// SIMATIC S7-200 SMART project (STEP 7-Micro/WIN SMART), CPU SR40

SYMBOL_TABLE 系统符号
Always_On        SM0.0    // 始终接通
First_Scan_On    SM0.1    // 仅在第一个扫描周期时接通
HSC0_Ctrl        SMB37    // 组态和控制 HSC0
HSC0_CV          SMD38    // HSC0 新当前值
HSC0_PV          SMD42    // HSC0 新预设值
END_SYMBOL_TABLE

ORGANIZATION_BLOCK MAIN:OB1
TITLE=程序注释
BEGIN
Network 1
// 程序段注释
LD     First_Scan_On:SM0.1
CALL   HSC0_INIT:SBR1
Network 2
LD     Always_On:SM0.0
=      L60.0
LD     I0.1
=      L63.7
LD     L60.0
CALL   PWM0_RUN:SBR2, L63.7, 1000, 500, VB10
END_ORGANIZATION_BLOCK

SUBROUTINE_BLOCK HSC0_INIT:SBR1
TITLE=
BEGIN
Network 1
// 要在程序内启用该组态，请使用 SM0.1 或沿触发指令从 MAIN 程序块将该子程序调用一次。  
// 针对模式 0 组态 HC0； CV = 0； PV = 4000； 加计数； 
// 将中断 COUNT_EQ0 附加到事件 12 (HC0 的 CV = PV)。
// 启用中断并启动计数器。
// 
LD     Always_On:SM0.0
MOVB   16#F8, HSC0_Ctrl:SMB37 //置位控制位： 加计数； 已启用； 
MOVD   +0, HSC0_CV:SMD38     //装载 CV
MOVD   +4000, HSC0_PV:SMD42  //装载 PV
HDEF   0, 0
ATCH   COUNT_EQ0:INT1, 12    //中断 COUNT_EQ0：HC0 的 CV = PV
ENI
HSC    0
SI     Q0.1, 1
RI     Q0.2, 1
END_SUBROUTINE_BLOCK

// SBR2: protected block, not included

INTERRUPT_BLOCK COUNT_EQ0:INT1
TITLE=
BEGIN
Network 1
// (CV = PV) 步 1，3，HC0
// 编译 HC0 的动态参数； PV = 7000； 
// 将中断 HSC0_STEP1 附加到事件 12 (HC0 的 CV = PV)。
// 启动计数器。
// 
LD     Always_On:SM0.0
MOVB   16#A0, HSC0_Ctrl:SMB37 //置位控制位： 写入预设值； 
MOVD   +7000, HSC0_PV:SMD42  //PV = 7000； 
ATCH   HSC0_STEP1:INT2, 12   //中断 HSC0_STEP1：HC0 的 CV = PV
HSC    0
SI     Q0.2, 1
END_INTERRUPT_BLOCK

INTERRUPT_BLOCK HSC0_STEP1:INT2
TITLE=
BEGIN
Network 1
// (CV = PV) 步 2，3，HC0
// 编译 HC0 的动态参数； PV = 3000； 减计数； 
// 将中断 HSC0_STEP2 附加到事件 12 (HC0 的 CV = PV)。
// 启动计数器。
// 
LD     Always_On:SM0.0
MOVB   16#B0, HSC0_Ctrl:SMB37 //置位控制位： 写入预设值； 减计数； 
MOVD   +3000, HSC0_PV:SMD42  //PV = 3000； 
ATCH   HSC0_STEP2:INT3, 12   //中断 HSC0_STEP2：HC0 的 CV = PV
HSC    0
RI     Q0.1, 1
END_INTERRUPT_BLOCK

INTERRUPT_BLOCK HSC0_STEP2:INT3
TITLE=
BEGIN
Network 1
// (CV = PV) 步 3，3，HC0
// 编译 HC0 的动态参数； CV = 0； PV = 4000； 加计数； 
// 将中断 COUNT_EQ0 附加到事件 12 (HC0 的 CV = PV)。
// 启动计数器。
// 
LD     Always_On:SM0.0
MOVB   16#F8, HSC0_Ctrl:SMB37 //置位控制位： 写入当前值； 写入预设值； 加计数； 
MOVD   +0, HSC0_CV:SMD38     //CV = 0； 
MOVD   +4000, HSC0_PV:SMD42  //PV = 4000； 
ATCH   COUNT_EQ0:INT1, 12    //中断 COUNT_EQ0：HC0 的 CV = PV
HSC    0
SI     Q0.1, 1
RI     Q0.2, 1
END_INTERRUPT_BLOCK
